TEXTLIST MoversMode_txt
  1 = 'Single'
  2 = 'Double'
  3 = 'Triple'
   = ''
END_TEXTLIST

(* stored: Version 1.1.0.1, ProductVersion 3.1.4024.11
   TextList MoversMode_txt: Id {50f0d7a1-51d1-4821-acbc-349e09e6ef3a} *)
